FUNCTION FC_Test : BOOL
VAR_INPUT
END_VAR
VAR
	temp_value: BOOL := False;
END_VAR




temp_value := GVL_VCM.test_bool_2;

GVL_VCM.test_bool_1 := temp_value;
temp_value := NOT GVL_VCM.test_bool_1;
GVL_VCM.test_bool_2 := temp_value;

RETURN;

END_FUNCTION

(* stored: Version 1.1.0.1, ProductVersion 3.1.4024.12
   POU FC_Test: Id {dcdc8aa2-9446-4cdf-b967-172534eff99c}, SpecialFunc None *)
